INTERFACE I_XtsPart

METHOD GetCurrentError : UDINT
VAR_INPUT
END_VAR
END_METHOD

PROPERTY HasError : BOOL
GET
END_GET
END_PROPERTY

METHOD Is24VBusOK : BOOL
END_METHOD

METHOD Is48VBusOK : BOOL
END_METHOD

METHOD ResetPart : BOOL
END_METHOD

METHOD SetInSim : HRESULT
VAR_INPUT
END_VAR
END_METHOD

METHOD SetPartOriginTransform : BOOL
VAR_INPUT
	OriginTransform: Tc3_XTS_Utility.ST_OriginTransform;
END_VAR
END_METHOD

END_INTERFACE

(* stored: Version 1.1.0.1
   Itf I_XtsPart: Id {79728d50-0c5c-4ced-9546-66681745df5e}
   Method GetCurrentError: Id {7903d85b-fb75-4c9a-8606-29b5130c9d6a}
   Property HasError: Id {3ffc12c8-866b-44c4-898c-7d9325cf0ff0}
   Get Get: Id {70faffad-0039-4f70-9833-ebc8c15c9c40}
   Method Is24VBusOK: Id {500c1a0d-a9c2-44cc-a7f0-1636e31cb371}
   Method Is48VBusOK: Id {65d6ebc5-d4c7-4450-a659-11bf3882ab2b}
   Method ResetPart: Id {6cd3b4ca-ad47-4f23-a5e9-46a25492ff53}
   Method SetInSim: Id {c9eb2856-51f9-4b2b-8bd3-e7c7234a0028}
   Method SetPartOriginTransform: Id {2de4d845-cfb8-4557-b610-ba9d0390b496} *)
